{attribute 'GeneratedUsingTerminal: EL2595-0000-0019'}
{attribute addProperty BoxType "EL2595-0000-0019"}
{attribute addProperty Id "EtcSlaveTerminalBaseDOX_StatusAT %I*DOX_Status_F52B34D37DOX_ControlAT %Q*DOX_Control_75D5C9E23WcStateAT %I*WcState_9091E0EB2InfoDataAT %I*InfoData_32EB74EA10"}
{attribute addProperty CRC "1469492337"}
{attribute addProperty Size "22"}
TYPE EL2595_5796AC71 EXTENDS EtcSlaveTerminalBase :
STRUCT
	{attribute addProperty Name "DOX_Status"}
	DOX_Status : DOX_Status_F52B34D3;
	{attribute addProperty Name "DOX_Control"}
	DOX_Control : DOX_Control_75D5C9E2;
	{attribute addProperty Name "WcState"}
	WcState : WcState_9091E0EB;
	{attribute addProperty Name "InfoData"}
	InfoData : InfoData_32EB74EA;
END_STRUCT
END_TYPE

(* stored: Version 1.2.0.0, ProductVersion 3.1.4024.9
   DUT EL2595_5796AC71: Id {7859fe1a-e5e4-4537-b35d-10f6e9cac24a} *)
